FUNCTION_BLOCK fbStepSequencer
VAR_INPUT
	iInStep:		INT;	//Constant, the step which this block instance represents
	iInNextStep:	INT;	//Next step to go to when this step is done. Will be moved into iCurrentStep when bInStepDone is true
	bInStepDone:	BOOL;	//If true and iCurrentStep = iInStep, then we move to the next step.
	tInStepDelay:	TIME;	//Time between when the bInStepDone rises to when we move states, set to 0 to disable.
	bInStepMode:	BOOL;	//This input will pause the state machine at the completion of the current step until bInStepAdvance is set high. 
	bInStepAdvance:	BOOL;	//When the state machine is paused, this input will trigger the next step.
	bInit:			BOOL;	//Initializes the state machine to step iInitStep.
	iInitStep:		INT;	//Step that the machine will be initialized to when bInit is true. 
END_VAR
VAR_OUTPUT
	bOutEnterEvent:	BOOL;	//High for one scan when the state machine enters the state specified by iInStep for a single block usage.
	bOutExitEvent:	BOOL;	//High for one scan when the state machine leaves iInStep
	bOutPaused:		BOOL;	//Indicates if the sequencer is paused and waiting on a bInStepAdvance signal. 
	iOutCurrentStep:INT;	//Current state/step
END_VAR
VAR
	bNextStepCondition:BOOL;
	bMonitorState:BOOL;
	TONStepDelay:TON;
	
	tempbInStepDone:BOOL;
	tempbInStepAdvance:BOOL;
	tempbInStepMode:BOOL;
	temptInStepDelay:TIME;
	
	bBlipEnterEvent:BOOL;
	bBlipExitEvent: BOOL;
	tempiInitStep: INT;
END_VAR



IF  (iInStep = iOutCurrentStep) THEN
	
	(*Set bOutEnterEvent on first entry to state*)
	IF NOT bBlipEnterEvent THEN
		bBlipEnterEvent:=1;
		bOutEnterEvent:=1;
	ELSE
		bOutEnterEvent:=0;
	END_IF
	
	(*sample the input only when we are in current step as using the same instance function block*)
	temptInStepDelay:=tInStepDelay;				
	tempbInStepDone:=bInStepDone;
	tempbInStepAdvance:=bInStepAdvance;
	tempbInStepMode:=bInStepMode;
	tempiInitStep:=iInitStep;
	TONStepDelay.IN:=1;
	
	(*next step condition*)
	bNextStepCondition:=  TONStepDelay.Q AND(NOT(tempbInStepMode) OR (tempbInStepMode AND tempbInStepAdvance));
	
	(*step complete map transition*)
	IF bNextStepCondition THEN
		TONStepDelay.IN:=0;              // reset step delay timer
		bBlipEnterEvent:=0;             //reset the one shot control for enter event
		bOutExitEvent:=1;				//Set only for one cycle 
		iOutCurrentStep:=iInNextStep;	//transition
	END_IF
	
ELSE
	bOutExitEvent:=0;
END_IF

(*if binit received make initp step the state we move to*)
IF bInit THEN
		bInit:=0;
		iOutCurrentStep:=iInitStep;
END_IF

TONStepDelay(PT:=tInStepDelay);

END_FUNCTION_BLOCK

(* stored: Version 1.1.0.1, ProductVersion 3.1.4024.11
   POU fbStepSequencer: Id {8babe64d-6080-4eb6-874b-84824d287606}, SpecialFunc None *)
